FUNCTION_BLOCK Iter
VAR
	_nIter		: UDINT;
	_bFirstLoop	: BOOL := TRUE;
END_VAR

//FB_Init is always available implicitly and it is used primarily for initialization.
//The return value is not evaluated. For a specific influence, you can also declare the
//methods explicitly and provide additional code there with the standard initialization
//code. You can evaluate the return value.
METHOD FB_Init: BOOL
VAR_INPUT
    bInitRetains: BOOL; // TRUE: the retain variables are initialized (reset warm / reset cold)
    bInCopyCode: BOOL;  // TRUE: the instance will be copied to the copy code afterward (online change)

	nInit		: UDINT;  
END_VAR
_nIter := nInit;
END_METHOD

METHOD Get : UDINT
VAR_INPUT
END_VAR
Get := _nIter;
END_METHOD

METHOD Next : UDINT
VAR_INPUT
END_VAR
IF _bFirstLoop THEN
	_bFirstLoop := FALSE;
	Next := _nIter;
	RETURN;	
END_IF

_nIter := _nIter + 1;
Next := _nIter;
END_METHOD

METHOD Peek : UDINT
VAR_INPUT
END_VAR
Peek := _nIter + 1;
END_METHOD

METHOD PeekBack : UDINT
VAR_INPUT
END_VAR
PeekBack := _nIter - 1;
END_METHOD

METHOD Prev : UDINT
VAR_INPUT
END_VAR
IF _bFirstLoop THEN
	_bFirstLoop := FALSE;
	Prev := _nIter;
	RETURN;	
END_IF

_nIter := _nIter - 1;
Prev := _nIter;
END_METHOD

METHOD Set : UDINT
VAR_INPUT
	nNewValue	: UDINT;
END_VAR
_nIter := nNewValue;
_bFirstLoop	:= TRUE;
Set := _nIter;
END_METHOD

END_FUNCTION_BLOCK

(* stored: Version 1.1.0.1
   POU Iter: Id {6e6052b3-52f3-4e20-af41-05a7fb850153}, SpecialFunc None
   Method FB_init: Id {44326773-18cb-44ea-8375-98f4b15aecc5}
   Method Get: Id {6cbdf049-35a0-4651-b09e-860b42e8ebbf}
   Method Next: Id {14f3edfe-b094-4f2c-b215-2ae55a0c7ec9}
   Method Peek: Id {ce151484-05ec-4af8-aa1e-65827fcb3415}
   Method PeekBack: Id {3b1ae5a1-134d-4bda-9724-ad7880e3bf37}
   Method Prev: Id {4226f68a-b1f5-430f-ae1b-d68632fc6002}
   Method Set: Id {3e15ac79-9132-4f58-b1de-a81f84ccd08d} *)
